(* CoDeSys 2.3.9.37 project: Cap11_7.pro *)
(* Libraries: Standard.lib 4.10.05 12:14:46, IecSfc.lib 13.4.06 16:51:28 *)

(* Global variable list: Global_Variables *)
VAR_GLOBAL

 (* Entradas *)
	M: BOOL;

      (*Salidas*)
	Rojo: BOOL;    	(* Luz roja*)
	Amarillo:BOOL;	(* Luz amarilla *)
	Verde:BOOL;		(* Luz verde *)

END_VAR

(* POU PLC_PRG, SFC *)
PROGRAM PLC_PRG
VAR
    (* declaración  de contadores *)
	CONTA: CTU;
END_VAR
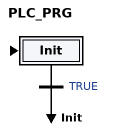
INITIAL_STEP Init:
END_STEP
TRANSITION FROM Init TO Init := TRUE;
END_TRANSITION
END_PROGRAM

(* Visualisation SemaforoSimple
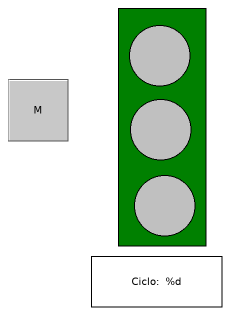
ellipse at (156,41)-(217,102): alarm colour if Rojo
ellipse at (157,115)-(218,176): alarm colour if Amarillo
ellipse at (161,191)-(222,252): alarm colour if Verde
rectangle at (118,272)-(249,323): text "Ciclo:  %d"; shows PLC_PRG.CONTA.CV
button at (35,95)-(95,157): text "M"; taps M
1 more shapes without text or variables
*)
